// Linearly interpolates between two values based on a given percentage.
FUNCTION F_Lerp : LREAL // The interpolated value.
VAR_INPUT
    fStartValue : LREAL; // The starting value.
    fEndValue   : LREAL; // The ending value.
    fPercentage : LREAL; // The interpolation factor (0.0 to 1.0).
END_VAR

F_Lerp := fStartValue + (fEndValue - fStartValue) * fPercentage;

END_FUNCTION

(* stored: Version 1.1.0.1
   POU F_Lerp: Id {8afff2ef-42b5-055b-15b3-074bf2e00bfb}, SpecialFunc None *)
